FUNCTION_BLOCK StringBuilderTests
VAR
    StringBuilder : TcoCore.StringBuilder();
    StringBuilderResult : STRING;
END_VAR

{attribute 'TcRpcEnable'}
METHOD Append
VAR_INPUT
    ToAppend : STRING;
END_VAR
StringBuilder.Append(ToAppend);
StringBuilderResult := StringBuilder._workString;
END_METHOD

{attribute 'TcRpcEnable'}
METHOD AppendAnyTest
StringBuilder.Clear();
// There was a strange compile-time error here... about function requiring exactly one input... could not get arround that... next time...
// 'AppendAny' is internal in the production code
//				     .AppendAny(_bool);
//					 .AppendAny(_real)
//					 .AppendAny(_lreal)
//					 .AppendAny(_dt)
//					 .AppendAny(_d)
//					 .AppendAny(_time)
//					 .AppendAny(_string)
//					 .AppendAny(_wstring)
//					 .AppendAny(_tod)
//					 .AppendAny(_int);
StringBuilderResult := StringBuilder._workString;
END_METHOD

{attribute 'TcRpcEnable'}
METHOD Clear
StringBuilder.Clear();
StringBuilderResult := StringBuilder._workString;
END_METHOD

{attribute 'TcRpcEnable'}
METHOD FluentApi : STRING
FluentApi :=
    StringBuilder.Clear().Append('1').Append('2').Append('3').Append('4').Clear().Append('1').Append('2').Append('3').Append('4').ToString();
END_METHOD

{attribute 'TcRpcEnable'}
METHOD ToString : STRING
ToString := StringBuilder.ToString();
StringBuilderResult := StringBuilder._workString;
END_METHOD

END_FUNCTION_BLOCK

(* stored: Version 1.1.0.1
   POU StringBuilderTests: Id {0281a88e-2ecd-0d34-1bf3-8e430317f9db}, SpecialFunc None
   Method Append: Id {f670e91a-c93f-018c-0969-450082bc795e}
   Method AppendAnyTest: Id {0674bf32-0aa6-01b8-156c-11f3869a6660}
   Method Clear: Id {164e99fa-4a83-04c8-2daa-d44516b3f0b2}
   Method FluentApi: Id {7518614b-0885-0114-1902-f5278e146ec7}
   Method ToString: Id {846c6a91-7892-0d0b-1eff-bbd62d279f18} *)
